KUKA KRL data list: vw_conv_usr_r.dat

&ACCESS RV
&PARAM DISKPATH = VW_User/Applikation/Conveyor
&PARAM TEMPLATE = C:\KRC\Roboter\Template\vw_usr_rv
&PARAM EDITMASK = vw_usr_r
&PARAM TPVW_VERSION = 8.3.18
&REL 139
DEFDAT VW_CONV_USR_R PUBLIC

;FOLD CONVEYORTECH GLOBALS
;
GLOBAL BOOL B_MIT_CONV=FALSE
;
;ENDFOLD (CONVEYORTECH GLOBALS)
ENDDAT
